// TIA Portal V18 export
TYPE "LGasp_MascheraCassetti"
// stored: IsFailsafeCompliant false
   STRUCT
      "name" : WString[30];   // nome del programma da PC
      ID : DInt;
      masking_1 : Array[1..16] of Bool;   // 1=presente
      masking_2 : Array[1..16] of Bool;   // 1=presente
      masking_3 : Array[1..16] of Bool;   // 1=presente
      masking_4 : Array[1..16] of Bool;   // 1=presente
   END_STRUCT;
END_TYPE
